(* delete old files and delete oldest files if number of files exceeds specified number *)
PROGRAM C09_MaintainFolders_OLD
VAR
	tArchiveCheck				: TIME := t#4s;
	fbMaintainArchive			: FB_PulseGenerator;
	tDeleteTimeCheck			: TIME := t#20m;
	fbMaintainDeleteTime		: FB_PulseGenerator;
	(*tDeleteItemCheck			: TIME := t#4s;
	fbMaintainDeleteItem		: FB_PulseGenerator;*)
	nActivateBitWord			: DWORD; (* if index increase 32 bits it is necceasry to declar 64 bits var like LREAL;*)

	aMaintainFolders			: ARRAY[1..17] OF NT_StartProcess;
	aManualMaintain			: ARRAY[1..17] OF BOOL;
	(*fbMoveOHMToArchive		: FB_OHM_MoveToArchive;*)
	(*fbMoveCACToArchive		: FB_CAC_MoveToArchive;*)
	fbMoveCHMToArchive		: FB_CHM_MoveToArchive;
	bZipCHMArchive			: BOOL;
	rtrigZipAfetrPassthrough		: R_TRIG;
	bManualZip					: BOOL;

	(*fbCompresOHMArchive		: NT_StartProcess;
	fbCompresCHMArchive		: NT_StartProcess;
	fbCompresPHMArchive		: NT_StartProcess;

	fbDeleteCHMNoLabel		: NT_StartProcess;*)

	fbRestoreTimer			: TON;
	fbRestoreOACFromCAC		: FB_CAC_RestoreOAC;
	nOCVFilesRestored			: UDINT;
	nOACFilesRestored			: UDINT;
	nCACFilesRestored			: UDINT;

	(*rtrigClearOCV				: R_TRIG;
	rtrigClearOCVError			: R_TRIG;
	rtrigClearOAC				: R_TRIG;
	rtrigClearOACError			: R_TRIG;

	fbClearOCVArchive			: FB_OCV_ClearArchive;
	fbClearOCVError			: FB_OCV_ClearArchive;
	fbClearOACArchive			: FB_OAC_ClearArchive;
	fbClearOACError			: FB_OAC_ClearArchive;

	rtrigClearOHM_FLG			: R_TRIG;
	rtrigClearCHM_FLG			: R_TRIG;

	fbClearOHM_FLG			: FB_OHM_ClearFLG;
	fbClearCHM_FLG			: FB_CHM_ClearFLG;
	btest : BOOL;*)

(********************************************************************************
		cBASE_FOLDER_ARR	: ARRAY[1..cSYSTEM_FOLDER_LIMIT] OF T_FolderName :=
			(*01*)'Bridge\',		(*02*)'Bridge\Archive\',		(*03*)'Bridge\Restore\',
			(*04*)'CAC\',		(*05*)'CAC\Archive\',		(*06*)'CAC\Error\',		(*07*)'CAC\Restore\', 	(*08*)'CAC\Restore\Archive\',
			(*09*)'CHM\',		(*10*)'CHM\Archive\',		(*11*)'CHM\Error\',		(*12*)'CHM\OK\',		(*13*)'CHM\Commissioning_Mode\',
			(*14*)'HMI\',
			(*15*)'KPI\',		(*16*)'KPI\Archive\',			(*17*)'KPI\Shift\',		(*18*)'KPI\ProdOrder\',
			(*19*)'OAC\',		(*20*)'OAC\Error\',
			(*21*)'OCV\',		(*22*)'OCV\Error\',
			(*23*)'OHM\',		(*24*)'OHM\Archive\',		(*25*)'OHM\Error\',		(*26*)'OHM\OK\',		(*27*)'OHM\Pending\',
			(*28*)'PCM\',		(*29*)'PCM\Archive\',		(*30*)'PCM\Error\',		(*31*)'PCM\Incoming\',
			(*32*)'PAC\',
			(*33*)'PHM\',		(*34*)'PHM\Archive\',		(*35*)'PHM\Error\',		(*36*)'PHM\OK\',
			(*37*)'Settings\',	(*38*)'Settings\Backups\',
			(*39*)'Templates\',
			(*40*)'Orca\',
			(*41*) 'SystemLog\';

*************************************************************************************)
(********************************************************************************
Delete Items
	DeleteItem <path> <filesToKeep> [createLog] [deleteDirs] [dirsToKeep]
	path: Directory path
	filesToKeep: Number OF files TO RETAIN
	createLog: (Optional) Boolean to enable logging
	deleteDirs: (Optional) Boolean to include directories
	dirsToKeep: (Optional) Number of directories to retain

Delete by Time
	DeleteTime <path> <fileAge> [createLog] [deleteDirs] [ageUnit]
	path: Directory path
	fileAge: Maximum age of files to retain
	createLog: (Optional) Boolean to enable logging
	deleteDirs: (Optional) Boolean to include inside directories for file search
	ageUnit: (Optional) Time unit for age values (Day/Hour/Minute), defaults to Day

Archive
	Archive <chmArchiveFolder> <lastArchiveDateName> [createLog]
	chmArchiveFolder: Archive folder path
	lastArchiveDateName: Last archive date identifier
	createLog: (Optional) Boolean TO enable logging
*************************************************************************************)
END_VAR

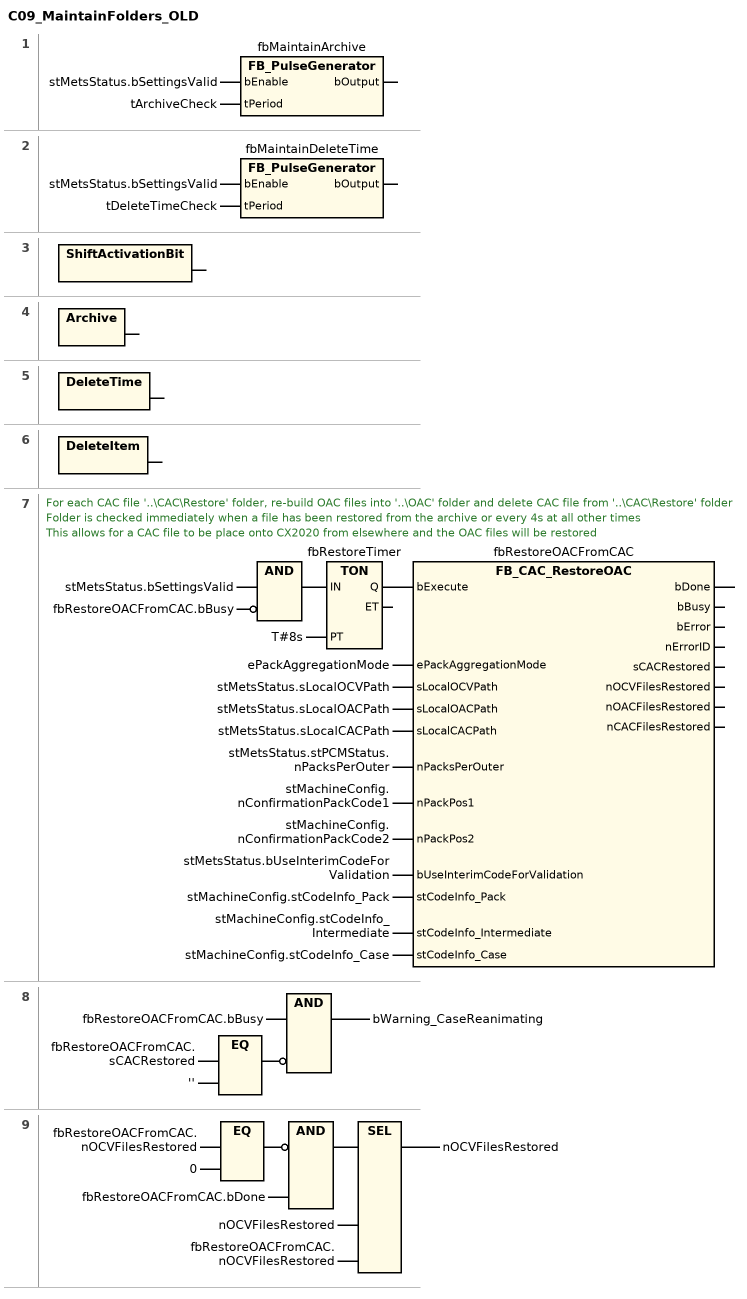
// NETWORK 1
fbMaintainArchive(bEnable := stMetsStatus.bSettingsValid, tPeriod := tArchiveCheck); // FB_PulseGenerator

// NETWORK 2
fbMaintainDeleteTime(bEnable := stMetsStatus.bSettingsValid, tPeriod := tDeleteTimeCheck); // FB_PulseGenerator

// NETWORK 3
ShiftActivationBit();

// NETWORK 4
Archive();

// NETWORK 5
DeleteTime();

// NETWORK 6
DeleteItem();

// NETWORK 7
// 					For each CAC file '..\CAC\Restore' folder, re-build OAC files into '..\OAC' folder and delete CAC file from '..\CAC\Restore' folder
// Folder is checked immediately when a file has been restored from the archive or every 4s at all other times
// This allows for a CAC file to be place onto CX2020 from elsewhere and the OAC files will be restored
//
fbRestoreTimer(IN := stMetsStatus.bSettingsValid AND NOT fbRestoreOACFromCAC.bBusy, PT := T#8s); // TON
fbRestoreOACFromCAC(
    bExecute := fbRestoreTimer.Q,
    ePackAggregationMode := ePackAggregationMode,
    sLocalOCVPath := stMetsStatus.sLocalOCVPath,
    sLocalOACPath := stMetsStatus.sLocalOACPath,
    sLocalCACPath := stMetsStatus.sLocalCACPath,
    nPacksPerOuter := stMetsStatus.stPCMStatus.nPacksPerOuter,
    nPackPos1 := stMachineConfig.nConfirmationPackCode1,
    nPackPos2 := stMachineConfig.nConfirmationPackCode2,
    bUseInterimCodeForValidation := stMetsStatus.bUseInterimCodeForValidation,
    stCodeInfo_Pack := stMachineConfig.stCodeInfo_Pack,
    stCodeInfo_Intermediate := stMachineConfig.stCodeInfo_Intermediate,
    stCodeInfo_Case := stMachineConfig.stCodeInfo_Case); // FB_CAC_RestoreOAC

// NETWORK 8
bWarning_CaseReanimating := fbRestoreOACFromCAC.bBusy AND NOT (fbRestoreOACFromCAC.sCACRestored = '');

// NETWORK 9
nOCVFilesRestored := SEL(NOT (fbRestoreOACFromCAC.nOCVFilesRestored = 0) AND fbRestoreOACFromCAC.bDone, nOCVFilesRestored, fbRestoreOACFromCAC.nOCVFilesRestored);

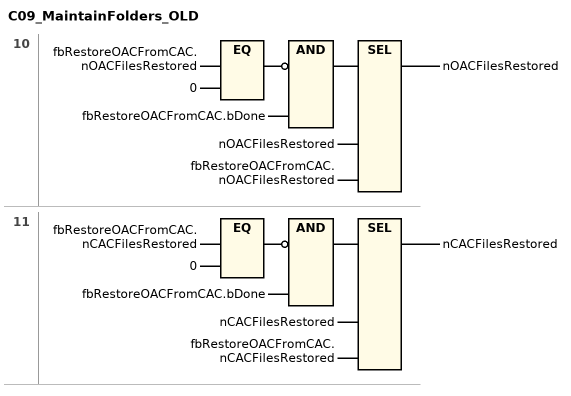
// NETWORK 10
nOACFilesRestored := SEL(NOT (fbRestoreOACFromCAC.nOACFilesRestored = 0) AND fbRestoreOACFromCAC.bDone, nOACFilesRestored, fbRestoreOACFromCAC.nOACFilesRestored);

// NETWORK 11
nCACFilesRestored := SEL(NOT (fbRestoreOACFromCAC.nCACFilesRestored = 0) AND fbRestoreOACFromCAC.bDone, nCACFilesRestored, fbRestoreOACFromCAC.nCACFilesRestored);

ACTION Archive:
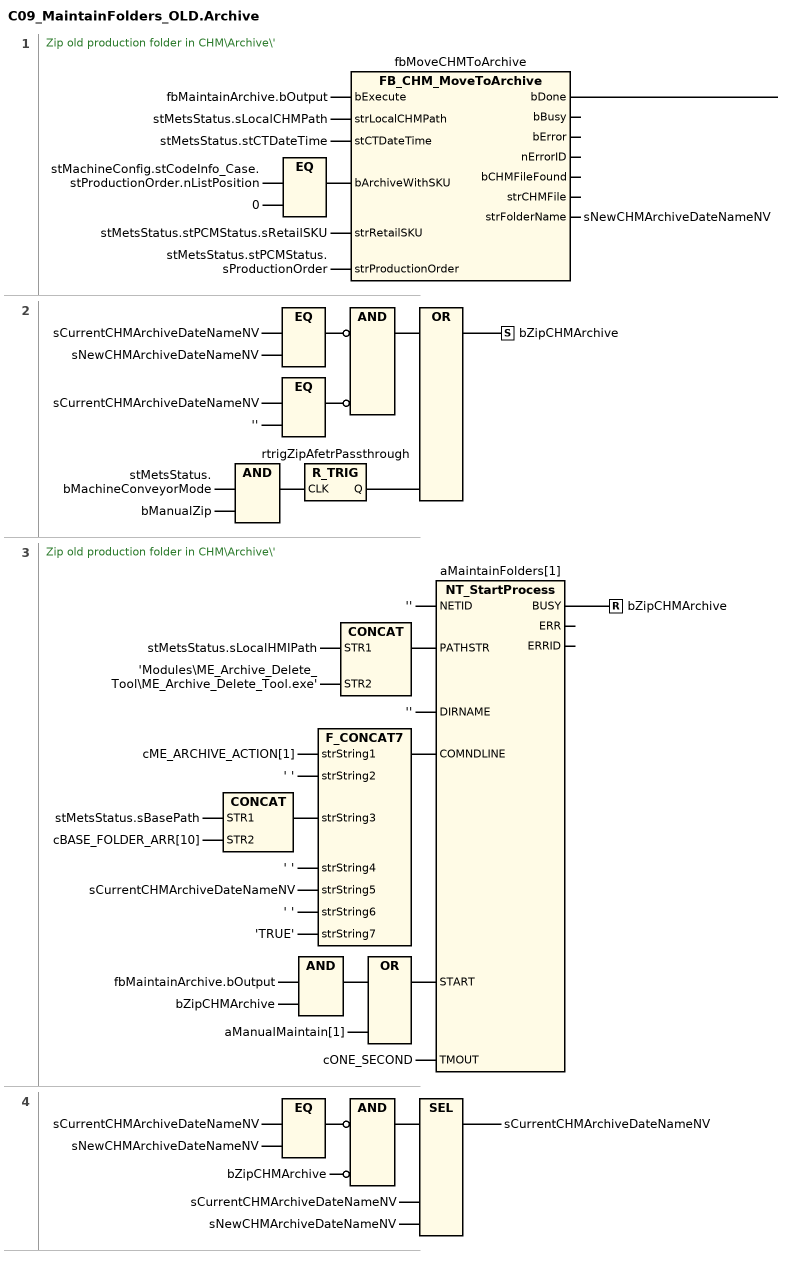
// NETWORK 1
// 					Zip old production folder in CHM\Archive\'
//
//
fbMoveCHMToArchive(
    bExecute := fbMaintainArchive.bOutput,
    strLocalCHMPath := stMetsStatus.sLocalCHMPath,
    stCTDateTime := stMetsStatus.stCTDateTime,
    bArchiveWithSKU := stMachineConfig.stCodeInfo_Case.stProductionOrder.nListPosition = 0,
    strRetailSKU := stMetsStatus.stPCMStatus.sRetailSKU,
    strProductionOrder := stMetsStatus.stPCMStatus.sProductionOrder,
    strFolderName => sNewCHMArchiveDateNameNV); // FB_CHM_MoveToArchive

// NETWORK 2
rtrigZipAfetrPassthrough(CLK := stMetsStatus.bMachineConveyorMode AND bManualZip); // R_TRIG
bZipCHMArchive S= NOT (sCurrentCHMArchiveDateNameNV = sNewCHMArchiveDateNameNV) AND NOT (sCurrentCHMArchiveDateNameNV = '') OR rtrigZipAfetrPassthrough.Q;

// NETWORK 3
// Zip old production folder in CHM\Archive\'
aMaintainFolders[1](
    NETID := '',
    PATHSTR := CONCAT(STR1 := stMetsStatus.sLocalHMIPath, STR2 := 'Modules\ME_Archive_Delete_Tool\ME_Archive_Delete_Tool.exe'),
    DIRNAME := '',
    COMNDLINE := F_CONCAT7(strString1 := cME_ARCHIVE_ACTION[1], strString2 := ' ', strString3 := CONCAT(STR1 := stMetsStatus.sBasePath, STR2 := cBASE_FOLDER_ARR[10]), strString4 := ' ', strString5 := sCurrentCHMArchiveDateNameNV, strString6 := ' ', strString7 := 'TRUE'),
    START := fbMaintainArchive.bOutput AND bZipCHMArchive OR aManualMaintain[1],
    TMOUT := cONE_SECOND); // NT_StartProcess
bZipCHMArchive R= aMaintainFolders[1].BUSY;

// NETWORK 4
sCurrentCHMArchiveDateNameNV := SEL(NOT (sCurrentCHMArchiveDateNameNV = sNewCHMArchiveDateNameNV) AND NOT bZipCHMArchive, sCurrentCHMArchiveDateNameNV, sNewCHMArchiveDateNameNV);
END_ACTION

ACTION DeleteItem:
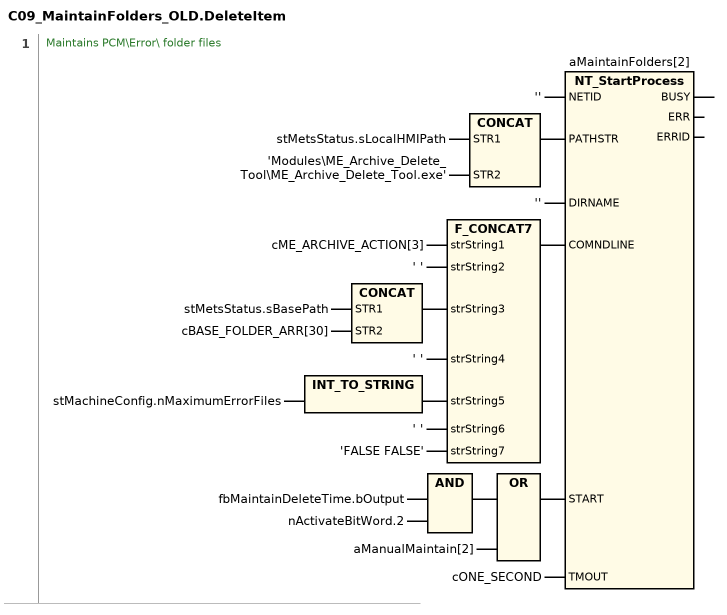
// NETWORK 1
// Maintains PCM\Error\ folder files
aMaintainFolders[2](
    NETID := '',
    PATHSTR := CONCAT(STR1 := stMetsStatus.sLocalHMIPath, STR2 := 'Modules\ME_Archive_Delete_Tool\ME_Archive_Delete_Tool.exe'),
    DIRNAME := '',
    COMNDLINE := F_CONCAT7(strString1 := cME_ARCHIVE_ACTION[3], strString2 := ' ', strString3 := CONCAT(STR1 := stMetsStatus.sBasePath, STR2 := cBASE_FOLDER_ARR[30]), strString4 := ' ', strString5 := INT_TO_STRING(stMachineConfig.nMaximumErrorFiles), strString6 := ' ', strString7 := 'FALSE FALSE'),
    START := fbMaintainDeleteTime.bOutput AND nActivateBitWord.2 OR aManualMaintain[2],
    TMOUT := cONE_SECOND); // NT_StartProcess

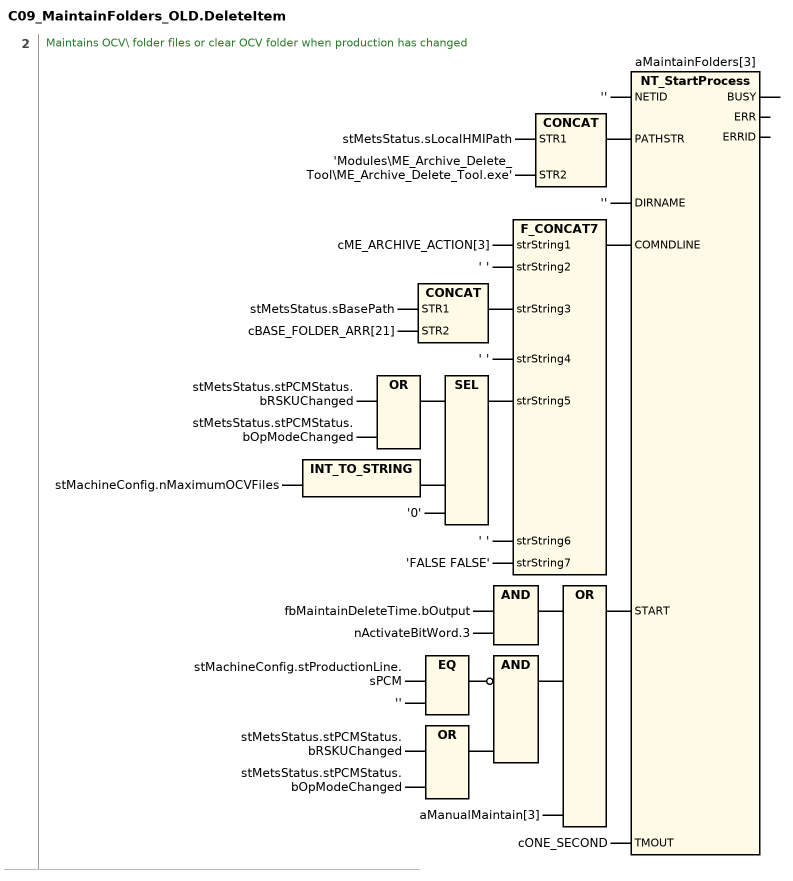
// NETWORK 2
// Maintains OCV\ folder files or clear OCV folder when production has changed
aMaintainFolders[3](
    NETID := '',
    PATHSTR := CONCAT(STR1 := stMetsStatus.sLocalHMIPath, STR2 := 'Modules\ME_Archive_Delete_Tool\ME_Archive_Delete_Tool.exe'),
    DIRNAME := '',
    COMNDLINE := F_CONCAT7(strString1 := cME_ARCHIVE_ACTION[3], strString2 := ' ', strString3 := CONCAT(STR1 := stMetsStatus.sBasePath, STR2 := cBASE_FOLDER_ARR[21]), strString4 := ' ', strString5 := SEL(stMetsStatus.stPCMStatus.bRSKUChanged OR stMetsStatus.stPCMStatus.bOpModeChanged, INT_TO_STRING(stMachineConfig.nMaximumOCVFiles), '0'), strString6 := ' ', strString7 := 'FALSE FALSE'),
    START := fbMaintainDeleteTime.bOutput AND nActivateBitWord.3 OR NOT (stMachineConfig.stProductionLine.sPCM = '') AND (stMetsStatus.stPCMStatus.bRSKUChanged OR stMetsStatus.stPCMStatus.bOpModeChanged) OR aManualMaintain[3],
    TMOUT := cONE_SECOND); // NT_StartProcess

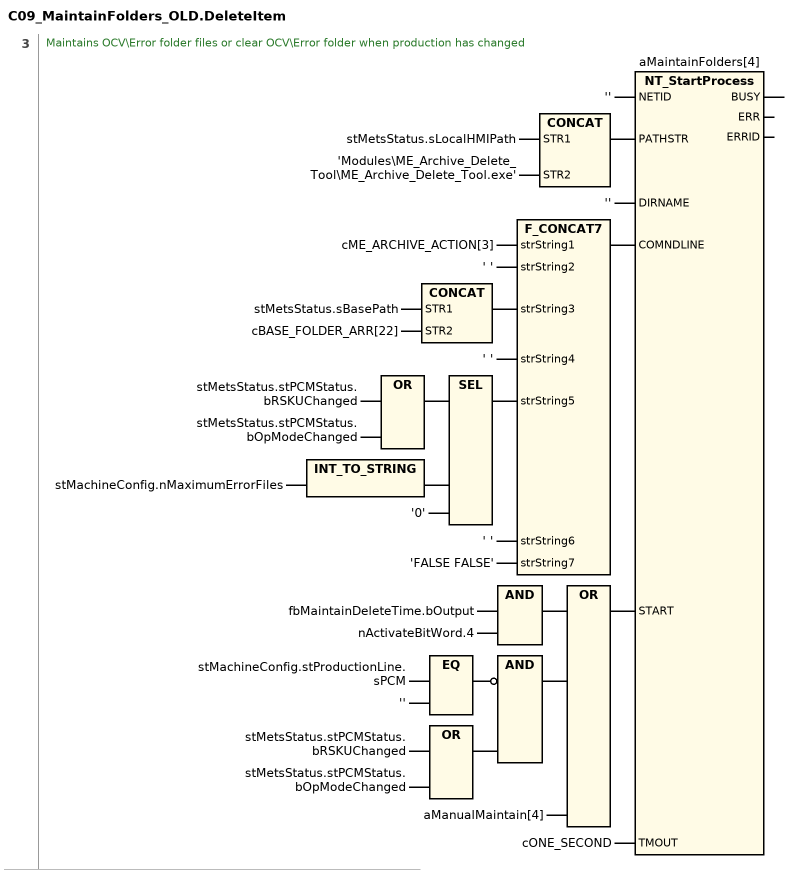
// NETWORK 3
// Maintains OCV\Error folder files or clear OCV\Error folder when production has changed
aMaintainFolders[4](
    NETID := '',
    PATHSTR := CONCAT(STR1 := stMetsStatus.sLocalHMIPath, STR2 := 'Modules\ME_Archive_Delete_Tool\ME_Archive_Delete_Tool.exe'),
    DIRNAME := '',
    COMNDLINE := F_CONCAT7(strString1 := cME_ARCHIVE_ACTION[3], strString2 := ' ', strString3 := CONCAT(STR1 := stMetsStatus.sBasePath, STR2 := cBASE_FOLDER_ARR[22]), strString4 := ' ', strString5 := SEL(stMetsStatus.stPCMStatus.bRSKUChanged OR stMetsStatus.stPCMStatus.bOpModeChanged, INT_TO_STRING(stMachineConfig.nMaximumErrorFiles), '0'), strString6 := ' ', strString7 := 'FALSE FALSE'),
    START := fbMaintainDeleteTime.bOutput AND nActivateBitWord.4 OR NOT (stMachineConfig.stProductionLine.sPCM = '') AND (stMetsStatus.stPCMStatus.bRSKUChanged OR stMetsStatus.stPCMStatus.bOpModeChanged) OR aManualMaintain[4],
    TMOUT := cONE_SECOND); // NT_StartProcess

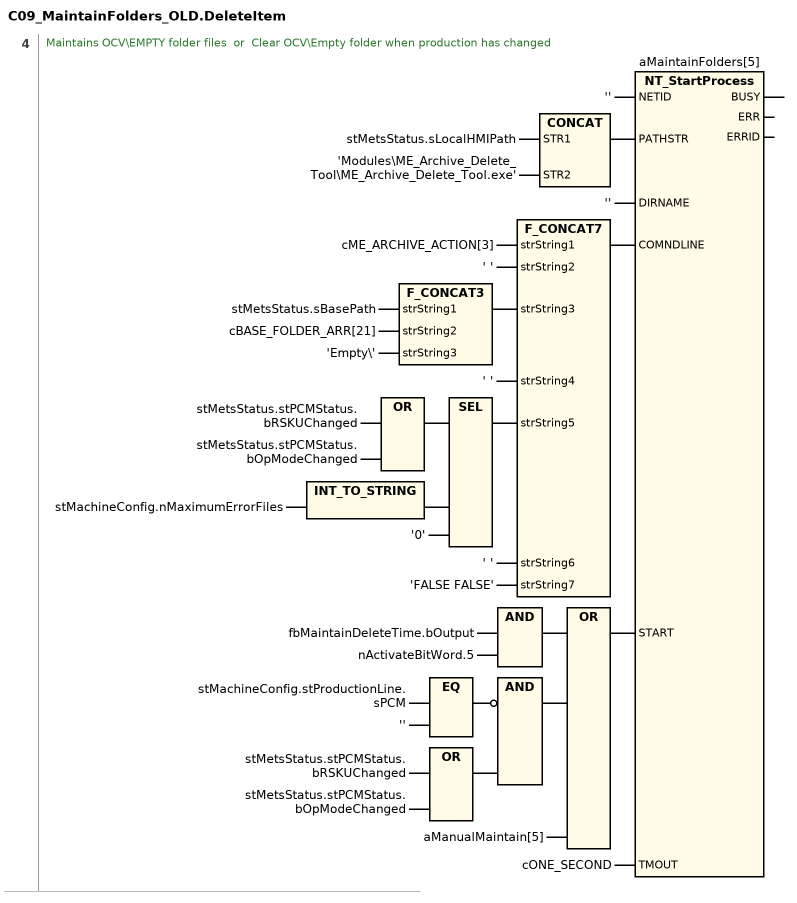
// NETWORK 4
// Maintains OCV\EMPTY folder files  or  Clear OCV\Empty folder when production has changed
aMaintainFolders[5](
    NETID := '',
    PATHSTR := CONCAT(STR1 := stMetsStatus.sLocalHMIPath, STR2 := 'Modules\ME_Archive_Delete_Tool\ME_Archive_Delete_Tool.exe'),
    DIRNAME := '',
    COMNDLINE := F_CONCAT7(strString1 := cME_ARCHIVE_ACTION[3], strString2 := ' ', strString3 := F_CONCAT3(strString1 := stMetsStatus.sBasePath, strString2 := cBASE_FOLDER_ARR[21], strString3 := 'Empty\'), strString4 := ' ', strString5 := SEL(stMetsStatus.stPCMStatus.bRSKUChanged OR stMetsStatus.stPCMStatus.bOpModeChanged, INT_TO_STRING(stMachineConfig.nMaximumErrorFiles), '0'), strString6 := ' ', strString7 := 'FALSE FALSE'),
    START := fbMaintainDeleteTime.bOutput AND nActivateBitWord.5 OR NOT (stMachineConfig.stProductionLine.sPCM = '') AND (stMetsStatus.stPCMStatus.bRSKUChanged OR stMetsStatus.stPCMStatus.bOpModeChanged) OR aManualMaintain[5],
    TMOUT := cONE_SECOND); // NT_StartProcess

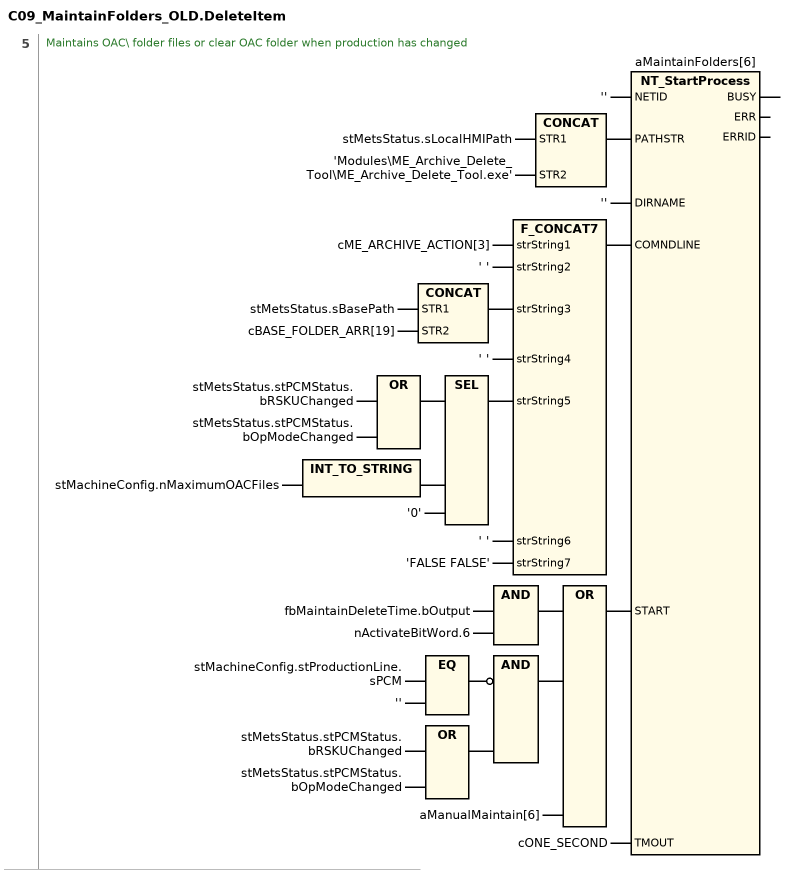
// NETWORK 5
// Maintains OAC\ folder files or clear OAC folder when production has changed
aMaintainFolders[6](
    NETID := '',
    PATHSTR := CONCAT(STR1 := stMetsStatus.sLocalHMIPath, STR2 := 'Modules\ME_Archive_Delete_Tool\ME_Archive_Delete_Tool.exe'),
    DIRNAME := '',
    COMNDLINE := F_CONCAT7(strString1 := cME_ARCHIVE_ACTION[3], strString2 := ' ', strString3 := CONCAT(STR1 := stMetsStatus.sBasePath, STR2 := cBASE_FOLDER_ARR[19]), strString4 := ' ', strString5 := SEL(stMetsStatus.stPCMStatus.bRSKUChanged OR stMetsStatus.stPCMStatus.bOpModeChanged, INT_TO_STRING(stMachineConfig.nMaximumOACFiles), '0'), strString6 := ' ', strString7 := 'FALSE FALSE'),
    START := fbMaintainDeleteTime.bOutput AND nActivateBitWord.6 OR NOT (stMachineConfig.stProductionLine.sPCM = '') AND (stMetsStatus.stPCMStatus.bRSKUChanged OR stMetsStatus.stPCMStatus.bOpModeChanged) OR aManualMaintain[6],
    TMOUT := cONE_SECOND); // NT_StartProcess

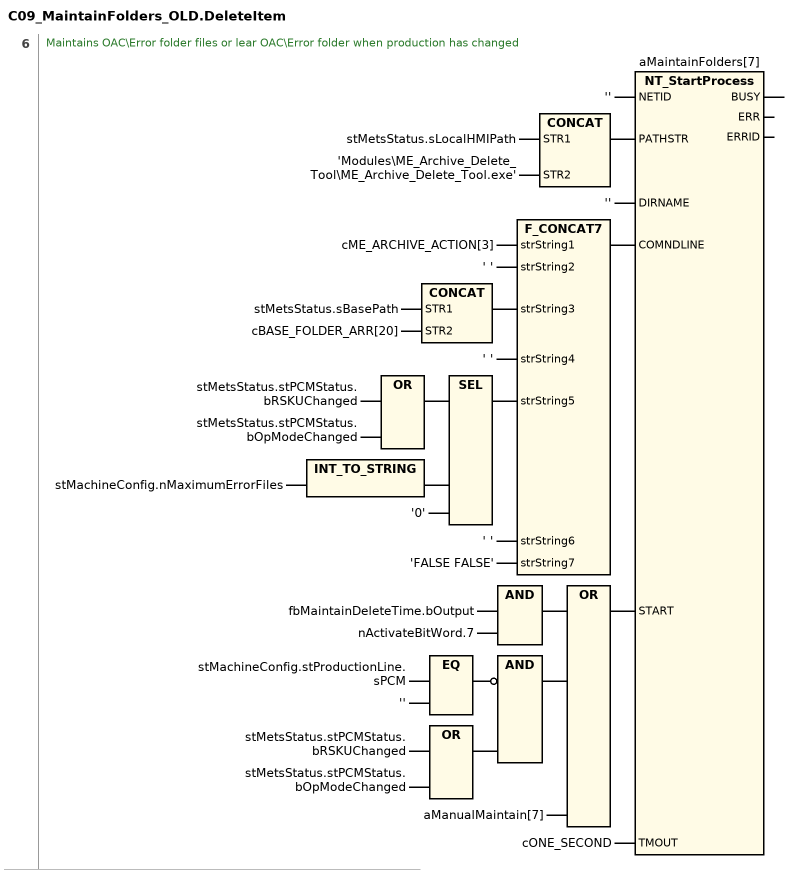
// NETWORK 6
// Maintains OAC\Error folder files or lear OAC\Error folder when production has changed
aMaintainFolders[7](
    NETID := '',
    PATHSTR := CONCAT(STR1 := stMetsStatus.sLocalHMIPath, STR2 := 'Modules\ME_Archive_Delete_Tool\ME_Archive_Delete_Tool.exe'),
    DIRNAME := '',
    COMNDLINE := F_CONCAT7(strString1 := cME_ARCHIVE_ACTION[3], strString2 := ' ', strString3 := CONCAT(STR1 := stMetsStatus.sBasePath, STR2 := cBASE_FOLDER_ARR[20]), strString4 := ' ', strString5 := SEL(stMetsStatus.stPCMStatus.bRSKUChanged OR stMetsStatus.stPCMStatus.bOpModeChanged, INT_TO_STRING(stMachineConfig.nMaximumErrorFiles), '0'), strString6 := ' ', strString7 := 'FALSE FALSE'),
    START := fbMaintainDeleteTime.bOutput AND nActivateBitWord.7 OR NOT (stMachineConfig.stProductionLine.sPCM = '') AND (stMetsStatus.stPCMStatus.bRSKUChanged OR stMetsStatus.stPCMStatus.bOpModeChanged) OR aManualMaintain[7],
    TMOUT := cONE_SECOND); // NT_StartProcess

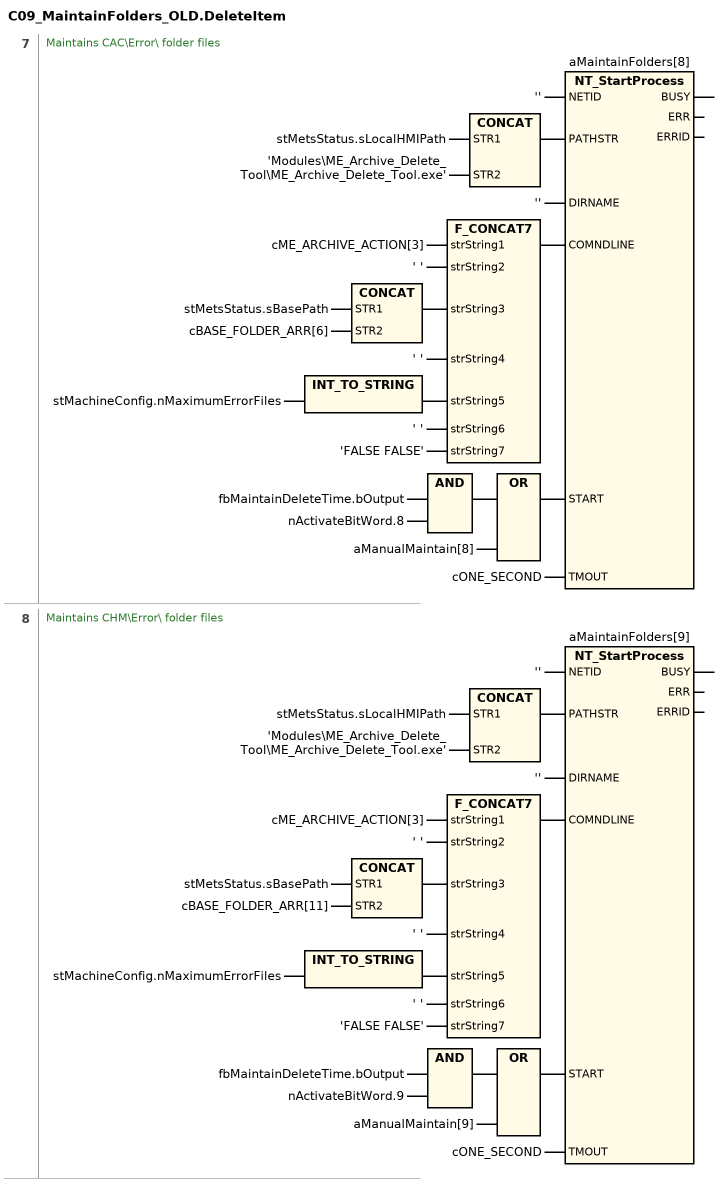
// NETWORK 7
// Maintains CAC\Error\ folder files
aMaintainFolders[8](
    NETID := '',
    PATHSTR := CONCAT(STR1 := stMetsStatus.sLocalHMIPath, STR2 := 'Modules\ME_Archive_Delete_Tool\ME_Archive_Delete_Tool.exe'),
    DIRNAME := '',
    COMNDLINE := F_CONCAT7(strString1 := cME_ARCHIVE_ACTION[3], strString2 := ' ', strString3 := CONCAT(STR1 := stMetsStatus.sBasePath, STR2 := cBASE_FOLDER_ARR[6]), strString4 := ' ', strString5 := INT_TO_STRING(stMachineConfig.nMaximumErrorFiles), strString6 := ' ', strString7 := 'FALSE FALSE'),
    START := fbMaintainDeleteTime.bOutput AND nActivateBitWord.8 OR aManualMaintain[8],
    TMOUT := cONE_SECOND); // NT_StartProcess

// NETWORK 8
// Maintains CHM\Error\ folder files
aMaintainFolders[9](
    NETID := '',
    PATHSTR := CONCAT(STR1 := stMetsStatus.sLocalHMIPath, STR2 := 'Modules\ME_Archive_Delete_Tool\ME_Archive_Delete_Tool.exe'),
    DIRNAME := '',
    COMNDLINE := F_CONCAT7(strString1 := cME_ARCHIVE_ACTION[3], strString2 := ' ', strString3 := CONCAT(STR1 := stMetsStatus.sBasePath, STR2 := cBASE_FOLDER_ARR[11]), strString4 := ' ', strString5 := INT_TO_STRING(stMachineConfig.nMaximumErrorFiles), strString6 := ' ', strString7 := 'FALSE FALSE'),
    START := fbMaintainDeleteTime.bOutput AND nActivateBitWord.9 OR aManualMaintain[9],
    TMOUT := cONE_SECOND); // NT_StartProcess

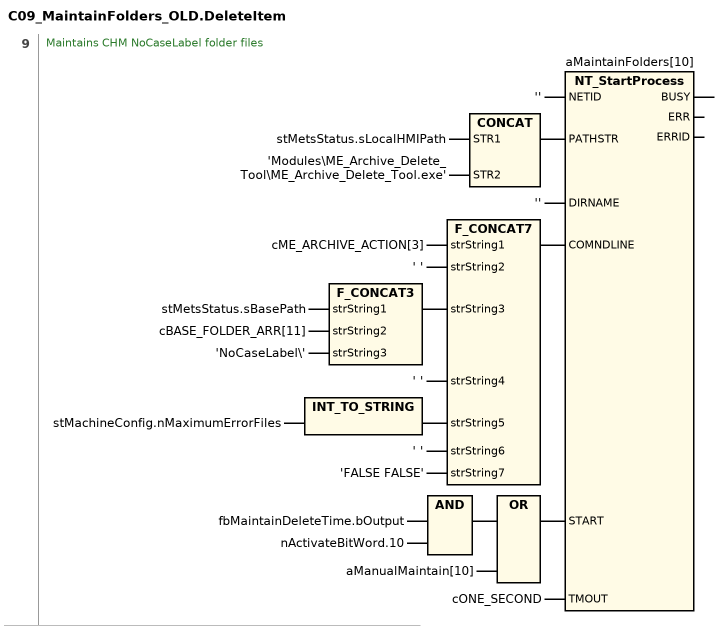
// NETWORK 9
// Maintains CHM NoCaseLabel folder files
aMaintainFolders[10](
    NETID := '',
    PATHSTR := CONCAT(STR1 := stMetsStatus.sLocalHMIPath, STR2 := 'Modules\ME_Archive_Delete_Tool\ME_Archive_Delete_Tool.exe'),
    DIRNAME := '',
    COMNDLINE := F_CONCAT7(strString1 := cME_ARCHIVE_ACTION[3], strString2 := ' ', strString3 := F_CONCAT3(strString1 := stMetsStatus.sBasePath, strString2 := cBASE_FOLDER_ARR[11], strString3 := 'NoCaseLabel\'), strString4 := ' ', strString5 := INT_TO_STRING(stMachineConfig.nMaximumErrorFiles), strString6 := ' ', strString7 := 'FALSE FALSE'),
    START := fbMaintainDeleteTime.bOutput AND nActivateBitWord.10 OR aManualMaintain[10],
    TMOUT := cONE_SECOND); // NT_StartProcess
END_ACTION

ACTION DeleteTime:
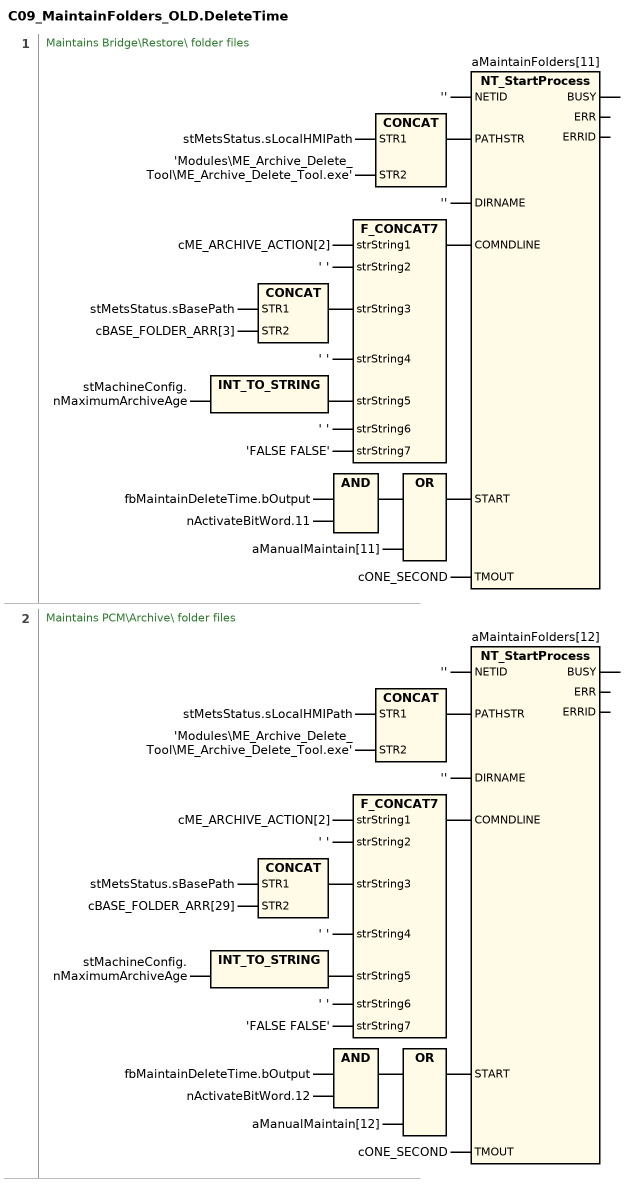
// NETWORK 1
// Maintains Bridge\Restore\ folder files
aMaintainFolders[11](
    NETID := '',
    PATHSTR := CONCAT(STR1 := stMetsStatus.sLocalHMIPath, STR2 := 'Modules\ME_Archive_Delete_Tool\ME_Archive_Delete_Tool.exe'),
    DIRNAME := '',
    COMNDLINE := F_CONCAT7(strString1 := cME_ARCHIVE_ACTION[2], strString2 := ' ', strString3 := CONCAT(STR1 := stMetsStatus.sBasePath, STR2 := cBASE_FOLDER_ARR[3]), strString4 := ' ', strString5 := INT_TO_STRING(stMachineConfig.nMaximumArchiveAge), strString6 := ' ', strString7 := 'FALSE FALSE'),
    START := fbMaintainDeleteTime.bOutput AND nActivateBitWord.11 OR aManualMaintain[11],
    TMOUT := cONE_SECOND); // NT_StartProcess

// NETWORK 2
// Maintains PCM\Archive\ folder files
aMaintainFolders[12](
    NETID := '',
    PATHSTR := CONCAT(STR1 := stMetsStatus.sLocalHMIPath, STR2 := 'Modules\ME_Archive_Delete_Tool\ME_Archive_Delete_Tool.exe'),
    DIRNAME := '',
    COMNDLINE := F_CONCAT7(strString1 := cME_ARCHIVE_ACTION[2], strString2 := ' ', strString3 := CONCAT(STR1 := stMetsStatus.sBasePath, STR2 := cBASE_FOLDER_ARR[29]), strString4 := ' ', strString5 := INT_TO_STRING(stMachineConfig.nMaximumArchiveAge), strString6 := ' ', strString7 := 'FALSE FALSE'),
    START := fbMaintainDeleteTime.bOutput AND nActivateBitWord.12 OR aManualMaintain[12],
    TMOUT := cONE_SECOND); // NT_StartProcess

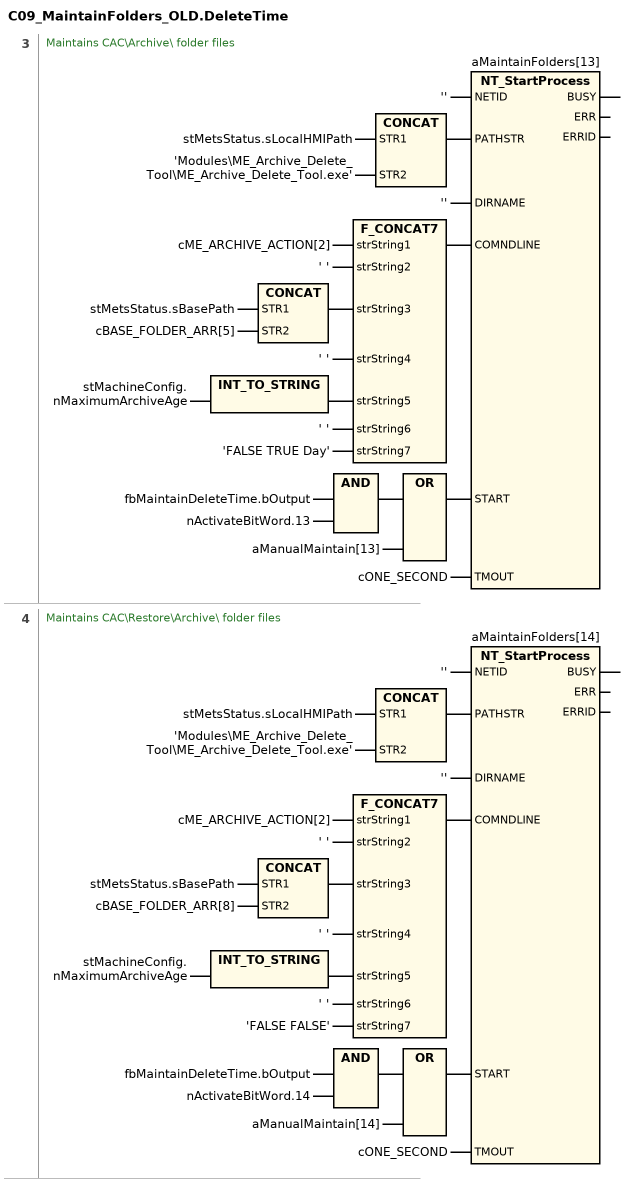
// NETWORK 3
// Maintains CAC\Archive\ folder files
aMaintainFolders[13](
    NETID := '',
    PATHSTR := CONCAT(STR1 := stMetsStatus.sLocalHMIPath, STR2 := 'Modules\ME_Archive_Delete_Tool\ME_Archive_Delete_Tool.exe'),
    DIRNAME := '',
    COMNDLINE := F_CONCAT7(strString1 := cME_ARCHIVE_ACTION[2], strString2 := ' ', strString3 := CONCAT(STR1 := stMetsStatus.sBasePath, STR2 := cBASE_FOLDER_ARR[5]), strString4 := ' ', strString5 := INT_TO_STRING(stMachineConfig.nMaximumArchiveAge), strString6 := ' ', strString7 := 'FALSE TRUE Day'),
    START := fbMaintainDeleteTime.bOutput AND nActivateBitWord.13 OR aManualMaintain[13],
    TMOUT := cONE_SECOND); // NT_StartProcess

// NETWORK 4
// Maintains CAC\Restore\Archive\ folder files
aMaintainFolders[14](
    NETID := '',
    PATHSTR := CONCAT(STR1 := stMetsStatus.sLocalHMIPath, STR2 := 'Modules\ME_Archive_Delete_Tool\ME_Archive_Delete_Tool.exe'),
    DIRNAME := '',
    COMNDLINE := F_CONCAT7(strString1 := cME_ARCHIVE_ACTION[2], strString2 := ' ', strString3 := CONCAT(STR1 := stMetsStatus.sBasePath, STR2 := cBASE_FOLDER_ARR[8]), strString4 := ' ', strString5 := INT_TO_STRING(stMachineConfig.nMaximumArchiveAge), strString6 := ' ', strString7 := 'FALSE FALSE'),
    START := fbMaintainDeleteTime.bOutput AND nActivateBitWord.14 OR aManualMaintain[14],
    TMOUT := cONE_SECOND); // NT_StartProcess

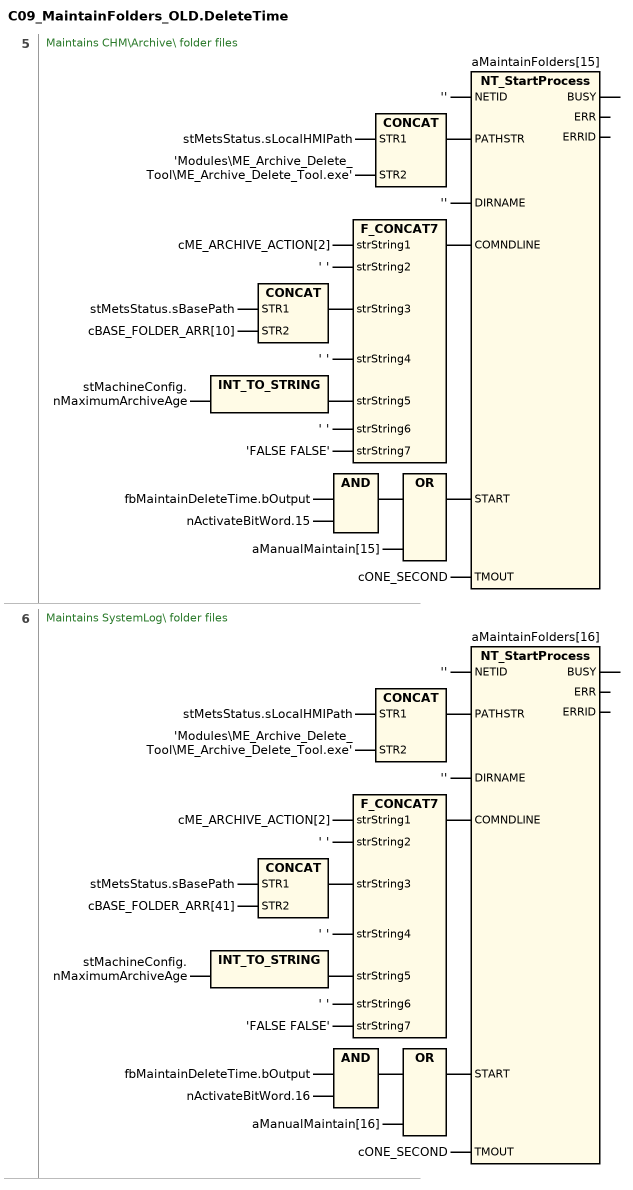
// NETWORK 5
// Maintains CHM\Archive\ folder files
aMaintainFolders[15](
    NETID := '',
    PATHSTR := CONCAT(STR1 := stMetsStatus.sLocalHMIPath, STR2 := 'Modules\ME_Archive_Delete_Tool\ME_Archive_Delete_Tool.exe'),
    DIRNAME := '',
    COMNDLINE := F_CONCAT7(strString1 := cME_ARCHIVE_ACTION[2], strString2 := ' ', strString3 := CONCAT(STR1 := stMetsStatus.sBasePath, STR2 := cBASE_FOLDER_ARR[10]), strString4 := ' ', strString5 := INT_TO_STRING(stMachineConfig.nMaximumArchiveAge), strString6 := ' ', strString7 := 'FALSE FALSE'),
    START := fbMaintainDeleteTime.bOutput AND nActivateBitWord.15 OR aManualMaintain[15],
    TMOUT := cONE_SECOND); // NT_StartProcess

// NETWORK 6
// Maintains SystemLog\ folder files
aMaintainFolders[16](
    NETID := '',
    PATHSTR := CONCAT(STR1 := stMetsStatus.sLocalHMIPath, STR2 := 'Modules\ME_Archive_Delete_Tool\ME_Archive_Delete_Tool.exe'),
    DIRNAME := '',
    COMNDLINE := F_CONCAT7(strString1 := cME_ARCHIVE_ACTION[2], strString2 := ' ', strString3 := CONCAT(STR1 := stMetsStatus.sBasePath, STR2 := cBASE_FOLDER_ARR[41]), strString4 := ' ', strString5 := INT_TO_STRING(stMachineConfig.nMaximumArchiveAge), strString6 := ' ', strString7 := 'FALSE FALSE'),
    START := fbMaintainDeleteTime.bOutput AND nActivateBitWord.16 OR aManualMaintain[16],
    TMOUT := cONE_SECOND); // NT_StartProcess

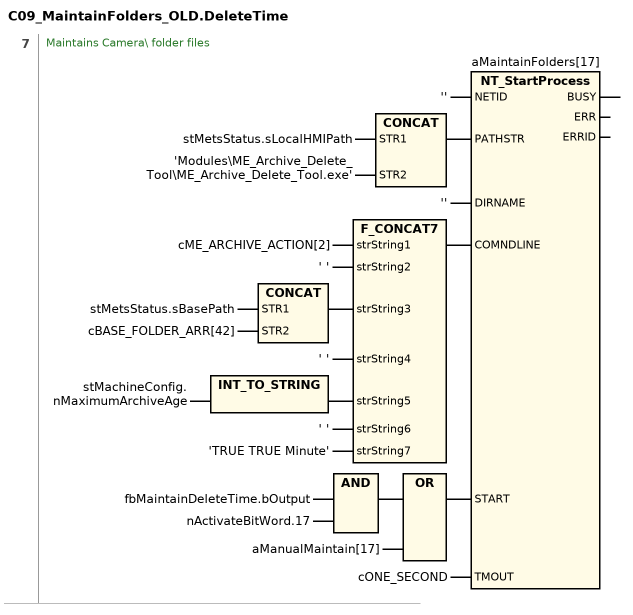
// NETWORK 7
// Maintains Camera\ folder files
aMaintainFolders[17](
    NETID := '',
    PATHSTR := CONCAT(STR1 := stMetsStatus.sLocalHMIPath, STR2 := 'Modules\ME_Archive_Delete_Tool\ME_Archive_Delete_Tool.exe'),
    DIRNAME := '',
    COMNDLINE := F_CONCAT7(strString1 := cME_ARCHIVE_ACTION[2], strString2 := ' ', strString3 := CONCAT(STR1 := stMetsStatus.sBasePath, STR2 := cBASE_FOLDER_ARR[42]), strString4 := ' ', strString5 := INT_TO_STRING(stMachineConfig.nMaximumArchiveAge), strString6 := ' ', strString7 := 'TRUE TRUE Minute'),
    START := fbMaintainDeleteTime.bOutput AND nActivateBitWord.17 OR aManualMaintain[17],
    TMOUT := cONE_SECOND); // NT_StartProcess
END_ACTION

ACTION ShiftActivationBit:
IF fbMaintainDeleteTime.bOutput	THEN
	IF nActivateBitWord = 0 THEN
		nActivateBitWord := 1;
	ELSE
		nActivateBitWord :=SHL(nActivateBitWord,1);
	END_IF
END_IF
END_ACTION

END_PROGRAM

(* stored: Version 1.1.0.1, ProductVersion 3.1.4024.15
   POU C09_MaintainFolders_OLD: Id {7cf7e03b-9fe9-4b11-be60-1bb8b5da7ce4}, SpecialFunc None
   Action Archive: Id {883d3b3c-6b7d-474d-bf9a-8d9ad0499434}
   Action DeleteItem: Id {f4d2e73f-3f57-4dba-a310-28e27cdfc175}
   Action DeleteTime: Id {cb7e326a-4106-4d6e-a544-06b2d74945cd}
   Action ShiftActivationBit: Id {b915070c-037f-4df1-98b4-f5aae29a4b88} *)
